// Mitsubishi GX Works2 project: TestComms   PLC: FX2N/FX2NC

PROGRAM MAIN
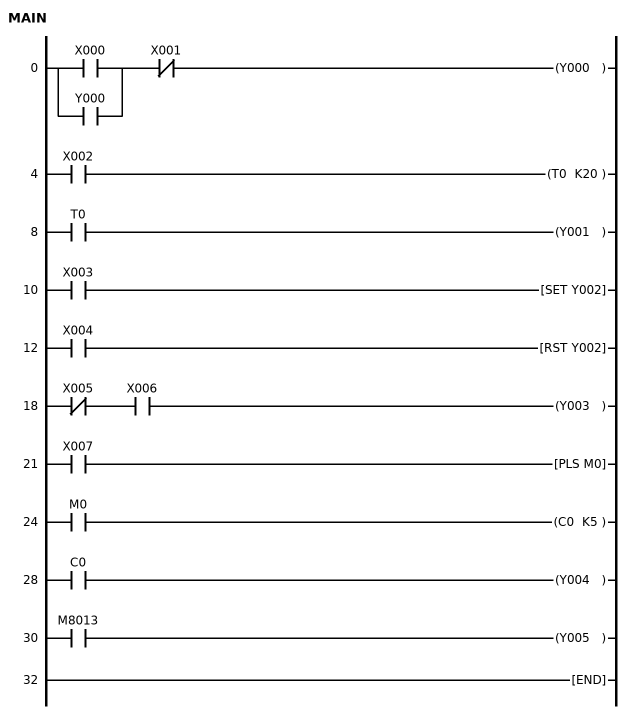
0     LD      X000
      OR      Y000
      ANI     X001
      OUT     Y000
4     LD      X002
      OUT     T0 K20
8     LD      T0
      OUT     Y001
10    LD      X003
      SET     Y002
12    LD      X004
      RST     Y002
18    LDI     X005
      AND     X006
      OUT     Y003
21    LD      X007
      PLS     M0
24    LD      M0
      OUT     C0 K5
28    LD      C0
      OUT     Y004
30    LD      M8013
      OUT     Y005
32    END
END_PROGRAM
